{attribute 'qualified_only'}
{attribute 'strict'}
TYPE E_Testcase :
(
	Stopped	:= -32768,
	Execute := 0,
	Done	:= 32767
)INT;
END_TYPE

(* stored: Version 1.1.0.1
   DUT E_Testcase: Id {6c594fbe-a1d3-4b2d-af82-ae3ef2090850} *)
